// Mitsubishi GX Works2 project: pr2.5   PLC: Q03UDV

PROGRAM MAIN
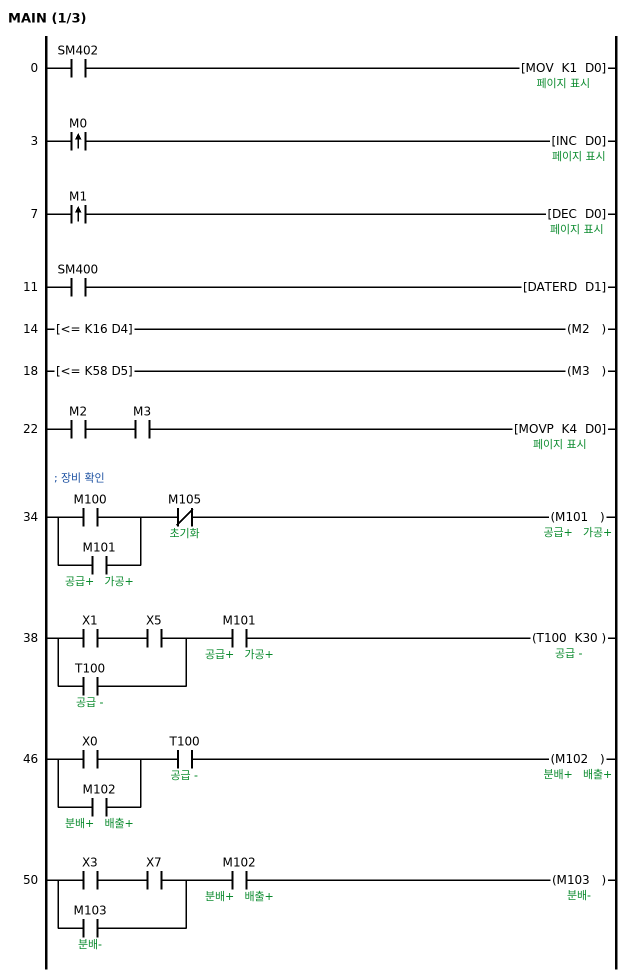
0     LD      SM402
      MOV     K1 D0  ; 페이지 표시
3     LDP     M0
      INC     D0
7     LDP     M1
      DEC     D0
11    LD      SM400
      DATERD  D1
14    LD<=    K16 D4
      OUT     M2
18    LD<=    K58 D5
      OUT     M3
22    LD      M2
      AND     M3
      MOVP    K4 D0
; 장비 확인
34    LD      M100
      OR      M101  ; 공급+   가공+
      ANI     M105  ; 초기화
      OUT     M101  ; 공급+   가공+
38    LD      X1
      AND     X5
      OR      T100  ; 공급 -
      AND     M101  ; 공급+   가공+
      OUT     T100 K30  ; 공급 -
46    LD      X0
      OR      M102  ; 분배+   배출+
      AND     T100  ; 공급 -
      OUT     M102  ; 분배+   배출+
50    LD      X3
      AND     X7
      OR      M103  ; 분배-
      AND     M102  ; 분배+   배출+
      OUT     M103  ; 분배-
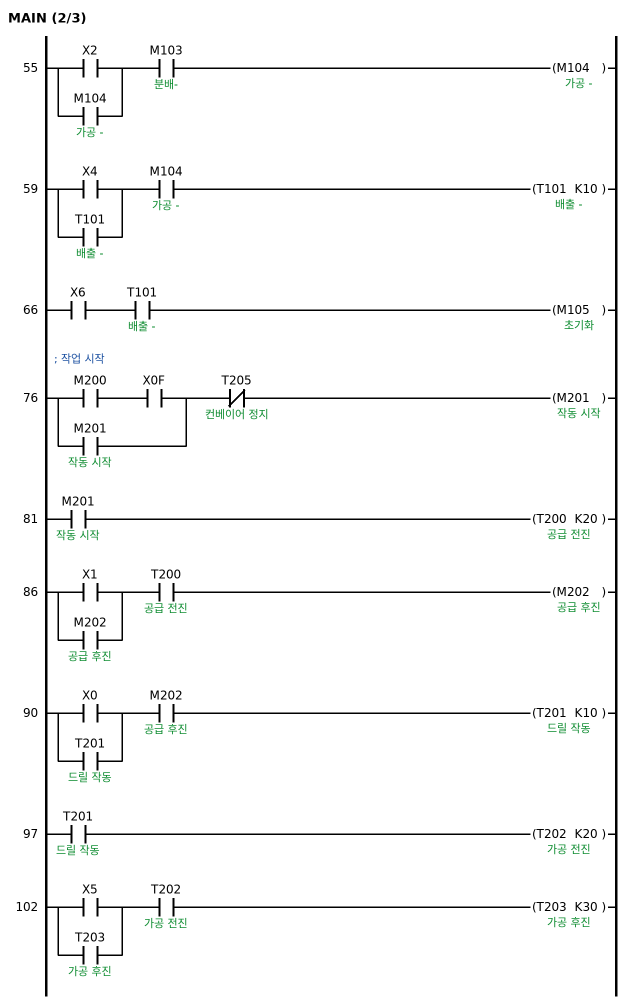
55    LD      X2
      OR      M104  ; 가공 -
      AND     M103  ; 분배-
      OUT     M104  ; 가공 -
59    LD      X4
      OR      T101  ; 배출 -
      AND     M104  ; 가공 -
      OUT     T101 K10  ; 배출 -
66    LD      X6
      AND     T101  ; 배출 -
      OUT     M105  ; 초기화
; 작업 시작
76    LD      M200
      AND     X0F
      OR      M201  ; 작동 시작
      ANI     T205  ; 컨베이어 정지
      OUT     M201  ; 작동 시작
81    LD      M201  ; 작동 시작
      OUT     T200 K20  ; 공급 전진
86    LD      X1
      OR      M202  ; 공급 후진
      AND     T200  ; 공급 전진
      OUT     M202  ; 공급 후진
90    LD      X0
      OR      T201  ; 드릴 작동
      AND     M202  ; 공급 후진
      OUT     T201 K10  ; 드릴 작동
97    LD      T201  ; 드릴 작동
      OUT     T202 K20  ; 가공 전진
102   LD      X5
      OR      T203  ; 가공 후진
      AND     T202  ; 가공 전진
      OUT     T203 K30  ; 가공 후진
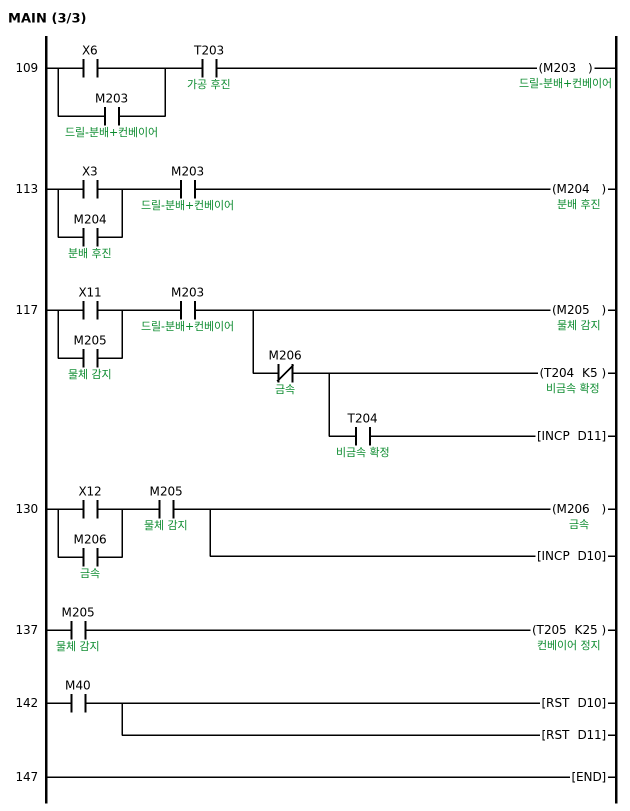
109   LD      X6
      OR      M203  ; 드릴-분배+컨베이어
      AND     T203  ; 가공 후진
      OUT     M203  ; 드릴-분배+컨베이어
113   LD      X3
      OR      M204  ; 분배 후진
      AND     M203  ; 드릴-분배+컨베이어
      OUT     M204  ; 분배 후진
117   LD      X11
      OR      M205  ; 물체 감지
      AND     M203  ; 드릴-분배+컨베이어
      OUT     M205  ; 물체 감지
      ANI     M206  ; 금속
      OUT     T204 K5  ; 비금속 확정
      AND     T204  ; 비금속 확정
      INCP    D11
130   LD      X12
      OR      M206  ; 금속
      AND     M205  ; 물체 감지
      OUT     M206  ; 금속
      INCP    D10
137   LD      M205  ; 물체 감지
      OUT     T205 K25  ; 컨베이어 정지
142   LD      M40
      RST     D10
      RST     D11
147   END
END_PROGRAM

PROGRAM OUTPUT
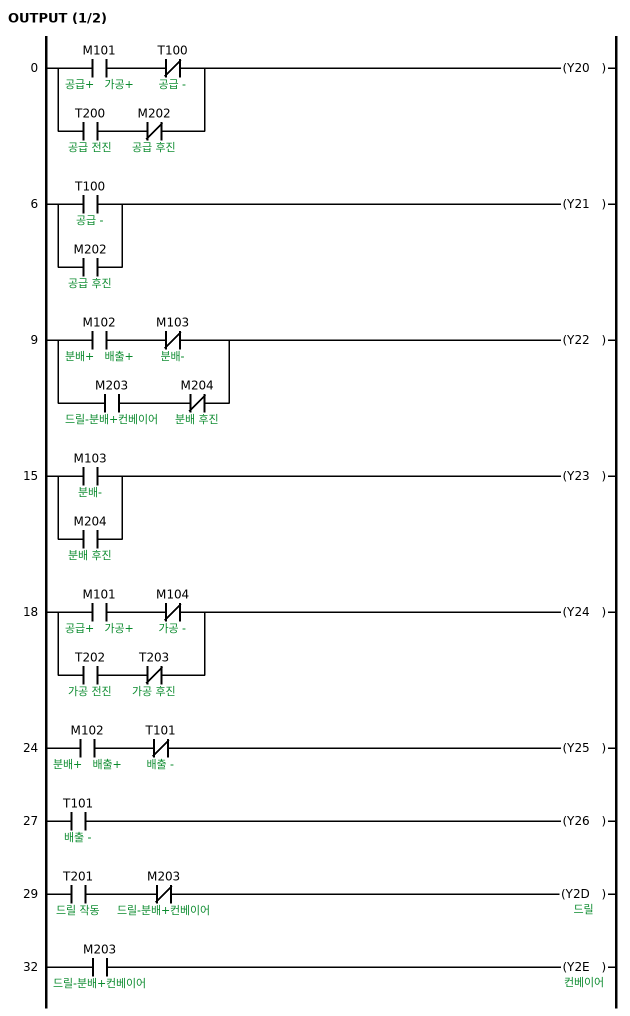
0     LD      M101  ; 공급+   가공+
      ANI     T100  ; 공급 -
      LD      T200  ; 공급 전진
      ANI     M202  ; 공급 후진
      ORB
      OUT     Y20
6     LD      T100  ; 공급 -
      OR      M202  ; 공급 후진
      OUT     Y21
9     LD      M102  ; 분배+   배출+
      ANI     M103  ; 분배-
      LD      M203  ; 드릴-분배+컨베이어
      ANI     M204  ; 분배 후진
      ORB
      OUT     Y22
15    LD      M103  ; 분배-
      OR      M204  ; 분배 후진
      OUT     Y23
18    LD      M101  ; 공급+   가공+
      ANI     M104  ; 가공 -
      LD      T202  ; 가공 전진
      ANI     T203  ; 가공 후진
      ORB
      OUT     Y24
24    LD      M102  ; 분배+   배출+
      ANI     T101  ; 배출 -
      OUT     Y25
27    LD      T101  ; 배출 -
      OUT     Y26
29    LD      T201  ; 드릴 작동
      ANI     M203  ; 드릴-분배+컨베이어
      OUT     Y2D  ; 드릴
32    LD      M203  ; 드릴-분배+컨베이어
      OUT     Y2E  ; 컨베이어
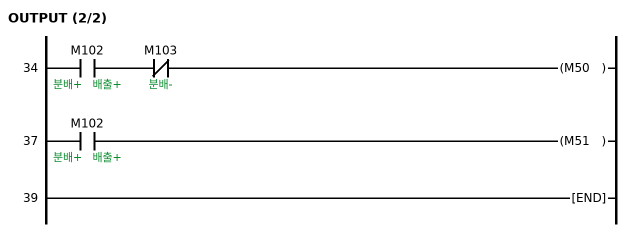
34    LD      M102  ; 분배+   배출+
      ANI     M103  ; 분배-
      OUT     M50
37    LD      M102  ; 분배+   배출+
      OUT     M51
39    END
END_PROGRAM

// device comments not shown above
X15  ; 회전
X16  ; 회전 정지
X20  ; 가 모 버
X21  ; 컨 모 버
X22  ; 공 전 버
X30  ; 컨 모 버
X40  ; 공 전 버
X41  ; 공 후 버
Y0D  ; 드릴
M10  ; 공급 시작
M11  ; 공급 +
M12  ; 공급 -
M13  ; 초기화
M20  ; 가공 모드
M21  ; 가공 +
M22  ; 가공-
M30  ; 분배 작동
M31  ; 분배 +
M32  ; 분배-
D3  ; \
